{attribute 'qualified_only'}
VAR_GLOBAL CONSTANT
  //Defect manager constants
	nMaxDefaults_C    							      : INT := 700; 
	nMaxDefaultsView_C   							    : INT := 20;
END_VAR

(* stored: Version 1.1.0.1, ProductVersion 3.1.4024.12
   GVL C: Id {b637d4a5-b39c-4bf9-8f55-3f1254518ed6} *)
